(* PLC project Unnamed, Unknown Unnamed 1 *)
(* stored: creationDateTime 2026-01-17T02:27:21, modificationDateTime 2026-01-17T02:27:21 *)

PROGRAM main
  VAR
    Temperature : INT := 22;
    Humidity : INT := 45;
    SetpointTemp : INT := 22;
    SetpointHumid : INT := 50;
    ChillerStatus : BOOL := FALSE;
    HumidifierStatus : BOOL := FALSE;
  END_VAR

            Temperature VAR INT %MW0 22
Humidity VAR INT %MW1 45
SetpointTemp VAR INT %MW2 22
SetpointHumid VAR INT %MW3 50
ChillerStatus VAR BOOL %QX0.0 FALSE
HumidifierStatus VAR BOOL %QX0.1 FALSE
          
END_PROGRAM

CONFIGURATION Config0
  RESOURCE Res0 ON PLC
    TASK task0(INTERVAL := T#20ms, PRIORITY := 1);
    PROGRAM instance0 WITH task0 : main;
  END_RESOURCE
END_CONFIGURATION
